FUNCTION_BLOCK FB_TCPModbusRequest_PV_Huawei_inclWrite_oneTurn
VAR_INPUT
	b_Enable: BOOL;
	by_slave_ID	:BYTE;
	str_IPAdress: STRING(15);
	uint_SetPoint_onetenth	:UINT;
END_VAR
VAR_OUTPUT

	lreal_RealPower_kW:LREAL;
	lreal_Voltage_L1L2_V: LREAL;
	lreal_Voltage_L2L3_V: LREAL;
	lreal_Voltage_L3L1_V: LREAL;
	lreal_Voltage_L1_V: LREAL;
	lreal_Voltage_L2_V: LREAL;
	lreal_Voltage_L3_V: LREAL;
	lreal_Current_L1_A: LREAL;
	lreal_Current_L2_A: LREAL;
	lreal_Current_L3_A: LREAL;
	lreal_PeakPowerDay_kW: LREAL;
	lreal_Power2_kW: LREAL;
	lreal_ReactivePower_kVAr: LREAL;
	lreal_PowerFactor: LREAL;
	lreal_Frequency_Hz: LREAL;
	lreal_Efficiency: LREAL;
	lreal_InternalTemperature_C: LREAL;
	lreal_IsolationResistance_MOhm: LREAL;
END_VAR
VAR
	i_State:INT;
	FB_SocketConnect : FB_SocketConnect;
	hSocket : T_HSOCKET;
	FB_SocketSend : FB_SocketSend;
	FB_SocketReceive : FB_SocketReceive;
	byteSendString : ARRAY[1..12] OF BYTE;
	FB_CloseSockets: FB_SocketCloseAll;
	
	ton_TimeOut: Ton;
	ton_WaitforReconnect: Ton;
	ton_ConnectionEstablised: Ton;
	time_ReconnectTime:TIME:=T#30M;
	byteReceiveString : ARRAY[1..200] OF BYTE;
	FB_BYTE_TO_WORD_1 : FB_CV_BYTE_TO_WORD;
	FB_BYTE_TO_WORD_2 : FB_CV_BYTE_TO_WORD;
	FB_WORD_TO_INT : FB_CV_WORD_TO_INT;
	ton_WaitforNetxtRequest: Ton;
	ton_Wait: Ton;
	int_SuccessCounter: INT;
	int_ReconnectCounter: INT;
	int_ErrorCount: INT;
	fbConvertWordToDword		: FB_CV_WORD_TO_DWORD;			//Convert Word to Dword
	fb_ConvertBytesToLreal		:fb_Convert4BytesToLreal;
	int_SuccessCounterWrite :INT;
	int_NotSuccessCounterWrite :INT;
	i	:INT;
	r_trig_Enable: R_trig;
	int_count: int;
	i_State_temp: INT;
	f_trig_Busy: f_trig;
	time_wait: TIME:= T#3S;
END_VAR


uint_SetPoint_onetenth := LIMIT (0,uint_SetPoint_onetenth,1000);



r_trig_Enable( clk := b_Enable);

CASE i_State OF
	0:	// wait for enable rising edge
		IF r_trig_Enable.Q THEN
			i_State := 1;
		END_IF
		FB_SocketConnect.bExecute := FALSE;
		FB_SocketSend.bExecute := FALSE;
		FB_SocketSend.bExecute := FALSE;
		ton_TimeOut.IN :=FALSE;	
		ton_ConnectionEstablised.IN := FALSE;
	

	1: // wait, not used now, old state
		i_State := i_State+1;
		
	2: // open socket
		FB_SocketConnect.bExecute := TRUE;
		ton_TimeOut.IN :=TRUE;
		i_State := i_State+1;
		
	3: // wait for connection established	
		IF NOT FB_SocketConnect.bBusy AND NOT FB_SocketConnect.bError THEN
			ton_TimeOut.IN :=FALSE;
			ton_ConnectionEstablised.IN := TRUE;
			i_State := i_State+1;
		ELSIF FB_SocketConnect.bError OR ton_TimeOut.Q THEN
			ton_TimeOut.IN :=FALSE;
			i_State := 100;
		END_IF
	
	4: //connection established, request data
		ton_Wait.IN := TRUE;
		// request FC3, Register 32064, 25 Words --> Real PV Power ff
		byteSendString[1] := 0;
		byteSendString[2] := 1;
		byteSendString[3] := 0;
		byteSendString[4] := 0;
		byteSendString[5] := 0;
		byteSendString[6] := 6;
		byteSendString[7] := LIMIT(1,by_slave_ID,255);			// slave id
		byteSendString[8] := 3;									// function code
		byteSendString[9] := 125;								// adress high
		byteSendString[10] := 64;								// adress low
		byteSendString[11] := 0;								// # of registers high
		byteSendString[12] := 25;								// # of registers low
		
		// clear receive buffer
		FOR i:= 1 TO 200 BY 1 DO
			byteReceiveString[i] := 0;
		END_FOR
		IF ton_Wait.Q THEN
			FB_SocketSend.bExecute := TRUE;
			ton_TimeOut.IN :=TRUE;
			ton_Wait.IN := FALSE;
			i_State := i_State+1;
		END_IF
	
	5: // wait for request sent
		IF NOT FB_SocketSend.bBusy AND NOT FB_SocketSend.bError THEN
			ton_TimeOut.IN :=FALSE;
			FB_SocketSend.bExecute := FALSE;
			i_State := i_State+1;  
		ELSIF FB_SocketSend.bError OR ton_TimeOut.Q THEN
			FB_SocketSend.bExecute := FALSE;
			ton_TimeOut.IN :=FALSE;
			i_State := 100;
		END_IF
		
	6: // wait for data
		ton_Wait.IN := TRUE;
		IF ton_Wait.Q THEN
			FB_SocketReceive.bExecute := TRUE;
			ton_Wait.IN := FALSE;
			i_State := i_State+1; 
		END_IF		 
	
	7:	
		ton_TimeOut.IN :=TRUE;
		IF f_trig_Busy.Q THEN
			FB_SocketReceive.bExecute := FALSE;
			i_State := i_State+1; 
		END_IF	
		IF ton_TimeOut.Q THEN
			FB_SocketReceive.bExecute := FALSE;
			ton_TimeOut.IN :=FALSE;
			i_State := 100;			
		END_IF
	
	8: // convert received data
		IF NOT FB_SocketReceive.bBusy AND NOT FB_SocketReceive.bError AND FB_SocketReceive.nRecBytes <> 0 THEN 
			int_SuccessCounter := int_SuccessCounter+1;
			ton_TimeOut.IN :=FALSE;
			FB_SocketReceive.bExecute := FALSE;
	
			FB_BYTE_TO_WORD_1(byInputValue_1 := byteReceiveString[14],byInputValue_2 := byteReceiveString[15], Ebyteorderforconvert := Ebyteorder.EBIGENDIAN, woutputvalue => );
			lreal_Voltage_L1L2_V := WORD_TO_LREAL(FB_BYTE_TO_WORD_1.woutputvalue)/10;
			FB_BYTE_TO_WORD_1(byInputValue_1 := byteReceiveString[16],byInputValue_2 := byteReceiveString[17], Ebyteorderforconvert := Ebyteorder.EBIGENDIAN, woutputvalue => );
			lreal_Voltage_L2L3_V := WORD_TO_LREAL(FB_BYTE_TO_WORD_1.woutputvalue)/10;
			FB_BYTE_TO_WORD_1(byInputValue_1 := byteReceiveString[18],byInputValue_2 := byteReceiveString[19], Ebyteorderforconvert := Ebyteorder.EBIGENDIAN, woutputvalue => );
			lreal_Voltage_L3L1_V := WORD_TO_LREAL(FB_BYTE_TO_WORD_1.woutputvalue)/10;
			FB_BYTE_TO_WORD_1(byInputValue_1 := byteReceiveString[20],byInputValue_2 := byteReceiveString[21], Ebyteorderforconvert := Ebyteorder.EBIGENDIAN, woutputvalue => );
			lreal_Voltage_L1_V := WORD_TO_LREAL(FB_BYTE_TO_WORD_1.woutputvalue)/10;
			FB_BYTE_TO_WORD_1(byInputValue_1 := byteReceiveString[22],byInputValue_2 := byteReceiveString[23], Ebyteorderforconvert := Ebyteorder.EBIGENDIAN, woutputvalue => );
			lreal_Voltage_L2_V := WORD_TO_LREAL(FB_BYTE_TO_WORD_1.woutputvalue)/10;
			FB_BYTE_TO_WORD_1(byInputValue_1 := byteReceiveString[24],byInputValue_2 := byteReceiveString[25], Ebyteorderforconvert := Ebyteorder.EBIGENDIAN, woutputvalue => );
			lreal_Voltage_L3_V := WORD_TO_LREAL(FB_BYTE_TO_WORD_1.woutputvalue)/10;


			fb_ConvertBytesToLreal(	by_InputValue_1:= byteReceiveString[10], 
									by_InputValue_2:= byteReceiveString[11], 
									by_InputValue_3:= byteReceiveString[12], 
									by_InputValue_4:= byteReceiveString[13], 
									int_Divider:= 1000, 
									lreal_Output=> );
					
			IF fb_ConvertBytesToLreal.lreal_Output < 100 AND fb_ConvertBytesToLreal.lreal_Output > -1 THEN
				lreal_RealPower_kW := fb_ConvertBytesToLreal.lreal_Output;
			END_IF
			
			fb_ConvertBytesToLreal(	by_InputValue_1:= byteReceiveString[26], 
									by_InputValue_2:= byteReceiveString[27], 
									by_InputValue_3:= byteReceiveString[28], 
									by_InputValue_4:= byteReceiveString[29], 
									int_Divider:= 1000, 
									lreal_Output=> lreal_Current_L1_A);
									
			fb_ConvertBytesToLreal(	by_InputValue_1:= byteReceiveString[30], 
									by_InputValue_2:= byteReceiveString[31], 
									by_InputValue_3:= byteReceiveString[32], 
									by_InputValue_4:= byteReceiveString[33], 
									int_Divider:= 1000, 
									lreal_Output=> lreal_Current_L2_A);

			fb_ConvertBytesToLreal(	by_InputValue_1:= byteReceiveString[34], 
									by_InputValue_2:= byteReceiveString[35], 
									by_InputValue_3:= byteReceiveString[36], 
									by_InputValue_4:= byteReceiveString[37], 
									int_Divider:= 1000, 
									lreal_Output=> lreal_Current_L3_A);
									
			fb_ConvertBytesToLreal(	by_InputValue_1:= byteReceiveString[38], 
									by_InputValue_2:= byteReceiveString[39], 
									by_InputValue_3:= byteReceiveString[40], 
									by_InputValue_4:= byteReceiveString[41], 
									int_Divider:= 1000, 
									lreal_Output=> lreal_PeakPowerDay_kW );

			fb_ConvertBytesToLreal(	by_InputValue_1:= byteReceiveString[42], 
									by_InputValue_2:= byteReceiveString[43], 
									by_InputValue_3:= byteReceiveString[44], 
									by_InputValue_4:= byteReceiveString[45], 
									int_Divider:= 1000, 
									lreal_Output=> lreal_Power2_kW);
			
			fb_ConvertBytesToLreal(	by_InputValue_1:= byteReceiveString[46], 
									by_InputValue_2:= byteReceiveString[47], 
									by_InputValue_3:= byteReceiveString[48], 
									by_InputValue_4:= byteReceiveString[49], 
									int_Divider:= 1000, 
									lreal_Output=>lreal_ReactivePower_kVAr );

			FB_BYTE_TO_WORD_1(byInputValue_1 := byteReceiveString[50],byInputValue_2 := byteReceiveString[51], Ebyteorderforconvert := Ebyteorder.EBIGENDIAN, woutputvalue => );
			lreal_PowerFactor := WORD_TO_LREAL(FB_BYTE_TO_WORD_1.woutputvalue)/1000;
			FB_BYTE_TO_WORD_1(byInputValue_1 := byteReceiveString[52],byInputValue_2 := byteReceiveString[53], Ebyteorderforconvert := Ebyteorder.EBIGENDIAN, woutputvalue => );
			lreal_Frequency_Hz := WORD_TO_LREAL(FB_BYTE_TO_WORD_1.woutputvalue)/100;
			FB_BYTE_TO_WORD_1(byInputValue_1 := byteReceiveString[54],byInputValue_2 := byteReceiveString[55], Ebyteorderforconvert := Ebyteorder.EBIGENDIAN, woutputvalue => );
			lreal_Efficiency := WORD_TO_LREAL(FB_BYTE_TO_WORD_1.woutputvalue)/100;
			FB_BYTE_TO_WORD_1(byInputValue_1 := byteReceiveString[56],byInputValue_2 := byteReceiveString[57], Ebyteorderforconvert := Ebyteorder.EBIGENDIAN, woutputvalue => );
			lreal_InternalTemperature_C := WORD_TO_LREAL(FB_BYTE_TO_WORD_1.woutputvalue)/10;
			FB_BYTE_TO_WORD_1(byInputValue_1 := byteReceiveString[58],byInputValue_2 := byteReceiveString[59], Ebyteorderforconvert := Ebyteorder.EBIGENDIAN, woutputvalue => );
			lreal_IsolationResistance_MOhm := WORD_TO_LREAL(FB_BYTE_TO_WORD_1.woutputvalue)/1000;

		
			//FB_WORD_TO_INT(wInputValue := FB_BYTE_TO_WORD.woutputvalue, iOutputValue => );
			//lreal_RealPower_kW := (INT_TO_LREAL(FB_WORD_TO_INT.iOutputValue))/1000;
			int_count := 0;
			i_State := i_State+1;
		ELSIF FB_SocketReceive.nRecBytes = 0 THEN
			
			IF int_count > 5 THEN
			 	i_State := 100;
				int_count := 0;
			ELSE
				i_State := 4;
				int_count := int_count + 1;
			END_IF	

(*		ELSIF FB_SocketSend.bError OR ton_TimeOut.Q THEN
 			FB_SocketReceive.bExecute := FALSE;
			ton_TimeOut.IN :=FALSE;
			i_State := 100;
*)		END_IF
	
	9: // for for next request
		IF FB_SocketReceive.nRecBytes = 0 THEN 
			i_State := 4;
		END_IF
		ton_WaitforNetxtRequest.IN := TRUE;
		IF ton_WaitforNetxtRequest.Q THEN
			ton_WaitforNetxtRequest.IN := FALSE;
			i_State := 20;
		END_IF
		IF 	ton_ConnectionEstablised.Q THEN 
			ton_WaitforNetxtRequest.IN := FALSE;
			i_State := 50;
		END_IF

	20: // write Setpoint
		ton_Wait.IN := TRUE;
		// request FC6 write register, Register 40125, 2 Word power setpoint
		byteSendString[1] := 0;
		byteSendString[2] := 1;
		byteSendString[3] := 0;
		byteSendString[4] := 0;
		byteSendString[5] := 0;
		byteSendString[6] := 6;
		byteSendString[7] := LIMIT(1,by_slave_ID,255);			// slave id
		byteSendString[8] := 6;									// function code
		byteSendString[9] := 156;								// adress high
		byteSendString[10] := 189;								// adress low
		byteSendString[11] := WORD_TO_BYTE(SHR(UINT_TO_WORD(uint_SetPoint_onetenth),8) AND 16#FFFF);		// # Value high
		byteSendString[12] := WORD_TO_BYTE(UINT_TO_WORD(uint_SetPoint_onetenth) AND 16#FFFF);				// # Value low		
	// clear receive buffer
		FOR i:= 1 TO 200 BY 1 DO
			byteReceiveString[i] := 0;
		END_FOR		
		IF ton_Wait.Q THEN
			FB_SocketSend.bExecute := TRUE;
			ton_TimeOut.IN :=TRUE;
			ton_Wait.IN := FALSE;
			i_State := i_State+1;
		END_IF
	
	21: // wait for request sent
		IF NOT FB_SocketSend.bBusy AND NOT FB_SocketSend.bError THEN
			ton_TimeOut.IN :=FALSE;
			FB_SocketSend.bExecute := FALSE;
			i_State := i_State+1;  
		ELSIF FB_SocketSend.bError OR ton_TimeOut.Q THEN
			FB_SocketSend.bExecute := FALSE;
			ton_TimeOut.IN :=FALSE;
			i_State := 100;
		END_IF		
		
	22: // wait for data
		ton_Wait.IN := TRUE;
		IF ton_Wait.Q THEN
			FB_SocketReceive.bExecute := TRUE;
			ton_Wait.IN := FALSE;
			i_State := i_State+1; 
		END_IF		 
	
	23:	
		ton_Wait.IN := TRUE;
		IF ton_Wait.Q THEN
			ton_TimeOut.IN :=TRUE;
			i_State := i_State+1; 
		END_IF	
	
	24: // Verify received data / writing succesful
		 	FB_SocketReceive.bExecute := FALSE;
		IF NOT FB_SocketReceive.bBusy AND NOT FB_SocketReceive.bError THEN
			
			IF 	byteReceiveString[5] = byteSendString[5] AND
				byteReceiveString[6] = byteSendString[6] AND
				byteReceiveString[7] = byteSendString[7] AND
				byteReceiveString[8] = byteSendString[8] AND 
				byteReceiveString[9] = byteSendString[9] AND
				byteReceiveString[10] = byteSendString[10] THEN
				int_SuccessCounterWrite := int_SuccessCounterWrite+1;
				i_State := i_State+1;
				int_count := 0;
			ELSE
				int_NotSuccessCounterWrite := int_NotSuccessCounterWrite+1;
				IF int_count > 5 THEN
				 	i_State := 100;
					int_count := 0;
				ELSE
					i_State := 20;
					int_count := int_count + 1;
				END_IF	
			END_IF
		

			
		ELSIF FB_SocketSend.bError OR ton_TimeOut.Q THEN
 			int_NotSuccessCounterWrite := int_NotSuccessCounterWrite+1;
			FB_SocketReceive.bExecute := FALSE;
			ton_TimeOut.IN :=FALSE;
			i_State := 100;
		END_IF
	
	25: // for for next request
		ton_WaitforNetxtRequest.IN := TRUE;
		IF ton_WaitforNetxtRequest.Q THEN
			ton_WaitforNetxtRequest.IN := FALSE;
			i_State := 50;
		END_IF
		IF 	ton_ConnectionEstablised.Q THEN 
			ton_WaitforNetxtRequest.IN := FALSE;
			i_State := 50;
		END_IF	
		
		
	50: // close sockets
		FB_CloseSockets.bExecute := TRUE;
		ton_TimeOut.IN :=TRUE;
		i_State := i_State+1;
		
	51: // wait for sockets closed
		
		IF NOT FB_CloseSockets.bBusy THEN
			int_ReconnectCounter := int_ReconnectCounter+1;
			FB_CloseSockets.bExecute := FALSE;
			i_State := 0;
		ELSIF FB_CloseSockets.bError THEN
			int_ReconnectCounter := int_ReconnectCounter+1;
			FB_CloseSockets.bExecute := FALSE;
			i_State := 0;
		END_IF

	100: // wait state for reconect
		
		FB_SocketConnect.bExecute := FALSE;
		FB_SocketSend.bExecute := FALSE;
		FB_SocketReceive.bExecute := FALSE;
		ton_ConnectionEstablised.IN := FALSE;
		ton_TimeOut.IN :=FALSE;
		ton_WaitforReconnect.IN := TRUE;
		IF ton_WaitforReconnect.Q THEN
			int_ErrorCount := int_ErrorCount+1;
			ton_WaitforReconnect.IN := FALSE;
			i_State := 50;
		END_IF
	
END_CASE
f_trig_Busy(clk := FB_SocketReceive.bBusy);


FB_SocketConnect(
	sSrvNetId := '',
	sRemoteHost := str_IPAdress,
	nRemotePort := 502,
	bExecute := ,
	tTimeout := T#5S,
	bBusy =>,
	bError =>,
	nErrId =>,
	hSocket => hSocket);
	
FB_SocketSend(
	sSrvNetId:= '', 
	hSocket:= hSocket, 
	cbLen:= 12,
	pSrc:= ADR( byteSendString ), 
	bExecute:= , 
	tTimeout:= T#5S, 
	bBusy=> , 
	bError=> , 
	nErrId=> );
	
FB_SocketReceive(
	sSrvNetId:= '', 
	hSocket:= hSocket, 
	cbLen:= 200, 
	pDest:= ADR( byteReceiveString ), 
	bExecute:= , 
	tTimeout:= T#5S, 
	bBusy=> , 
	bError=> , 
	nErrId=> , 
	nRecBytes=> );

FB_CloseSockets(
	sSrvNetId:= '', 
	bExecute:= , 
	tTimeout:= T#2S, 
	bBusy=> , 
	bError=> , 
	nErrId=> );
	
ton_TimeOut(PT := T#10S);
ton_WaitforReconnect(PT := T#10S);
ton_ConnectionEstablised(pt := time_ReconnectTime);
ton_WaitforNetxtRequest(PT:= T#2S);
ton_Wait(PT:=time_wait);

END_FUNCTION_BLOCK

(* stored: Version 1.1.0.1, ProductVersion 3.1.4024.12
   POU FB_TCPModbusRequest_PV_Huawei_inclWrite_oneTurn: Id {03cd1501-e5f6-4ac1-985d-500dbfd8b8d5}, SpecialFunc None *)
